# EPICS autosave request: SIS8300bpmApp/Db/SIS8300bpm_settings.req
$(P)$(R)NearIQM
$(P)$(R)NearIQN
$(P)$(R)MemMux
$(P)$(R)MemMux10
$(P)$(R)TrigSetup
$(P)$(R)FilterControl
$(P)$(R)FilterEnable
$(P)$(R)FilterCoeff0
$(P)$(R)FilterCoeff1
$(P)$(R)FilterCoeff2
$(P)$(R)FilterCoeff3
$(P)$(R)FilterCoeff4
$(P)$(R)FilterCoeff5
